ABB RobotStudio station: LAB1RS_20220902-140616.rsstn

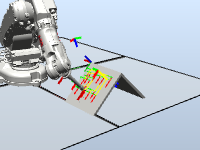
Station LAB1RS (saved by RobotStudio 6.5.7558.2005)
Controller IRB_140_6kg_0.81m
  mechanical unit ROB_1: IRB140_6_81_C_03, 6 joints, base frame (0, 0, 0) mm
Layout (positions relative to the parent item):
  - IRB140_6_81_C_03 [mechanism, from Robots\IRB140_6_81_C_G_03.rslib] at (0, 0, 0) mm; joint values [-0.1973, 1.0047, -0.2124, 0.8557, 1.1481, -2.2858] (rad or m)
  - TABLERO2 [part] at (800, 200, 0) mm, rotated rx 90 ry 0 rz 90 deg
  - TOOLSJ [mechanism, from Libraries\HCV2.rslib] at (628.25, -79.94, 228.26) mm, rotated rx 180 ry 44.6 rz -90 deg
Attachment: TOOLSJ is attached to IRB140_6_81_C_03 / Link6
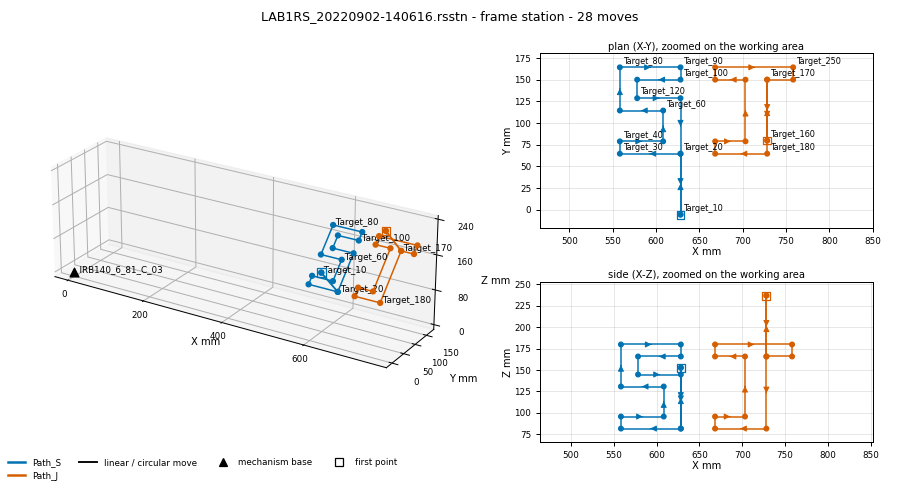
[picture p0: tool path of LAB1RS_20220902-140616.rsstn in frame station, 28 of 30 moves have a stored position in this frame; points joined in program order, loops and branches not executed]
Targets, tools, work objects and paths stored in the station, written as RAPID:
! task T_ROB1
MODULE CalibData
  TASK PERS wobjdata TabSJ:=[FALSE,TRUE,"",[[516.5,200,215],[0,0,-0.379480687,0.925199658]],[[0,0,0],[1,0,0,0]]];
  PERS tooldata HCVTCP:=[TRUE,[[0,0,191.01],[1,0,0,0]],[0.16,[0,0,75.29],[1,0,0,0],0,0,0]];
  PERS tooldata TOOLSJTCP:=[TRUE,[[0,0,191.01],[1,0,0,0]],[0.2,[0,0,1],[1,0,0,0],0,0,0]];
ENDMODULE

! task T_ROB1
MODULE Module1
  CONST jointtarget Home:=[[0,0,0,0,0,0],[9E+09,9E+09,9E+09,9E+09,9E+09,9E+09]];
  CONST jointtarget Mid:=[[0,30,0,0,30,0],[9E+09,9E+09,9E+09,9E+09,9E+09,9E+09]];
  CONST robtarget Target_10:=[[-111.75,190.000000035,99.999999935],[0,0.707106781,0.707106781,0],[0,0,0,0],[9E+09,9E+09,9E+09,9E+09,9E+09,9E+09]];
  CONST robtarget Target_20:=[[-111.75,190,-0.000000065],[0,0.707106781,0.707106781,0],[0,0,0,0],[9E+09,9E+09,9E+09,9E+09,9E+09,9E+09]];
  CONST robtarget Target_30:=[[-41.75,190,-0.000000065],[0,0.707106781,0.707106781,0],[0,0,0,0],[9E+09,9E+09,9E+09,9E+09,9E+09,9E+09]];
  CONST robtarget Target_40:=[[-41.75,170,-0.000000057],[0,0.707106781,0.707106781,0],[0,0,0,0],[9E+09,9E+09,9E+09,9E+09,9E+09,9E+09]];
  CONST robtarget Target_50:=[[-91.75,170,-0.000000057],[0,0.707106781,0.707106781,0],[0,0,0,0],[9E+09,9E+09,9E+09,9E+09,9E+09,9E+09]];
  CONST robtarget Target_60:=[[-91.75,120,-0.000000041],[0,0.707106781,0.707106781,0],[0,0,0,0],[9E+09,9E+09,9E+09,9E+09,9E+09,9E+09]];
  CONST robtarget Target_70:=[[-41.75,120,-0.000000041],[0,0.707106781,0.707106781,0],[0,0,0,0],[9E+09,9E+09,9E+09,9E+09,9E+09,9E+09]];
  CONST robtarget Target_80:=[[-41.75,50,-0.000000017],[0,0.707106781,0.707106781,0],[0,0,0,0],[9E+09,9E+09,9E+09,9E+09,9E+09,9E+09]];
  CONST robtarget Target_90:=[[-111.75,50,-0.000000017],[0,0.707106781,0.707106781,0],[0,0,0,0],[9E+09,9E+09,9E+09,9E+09,9E+09,9E+09]];
  CONST robtarget Target_100:=[[-111.75,70,-0.000000024],[0,0.707106781,0.707106781,0],[0,0,0,0],[9E+09,9E+09,9E+09,9E+09,9E+09,9E+09]];
  CONST robtarget Target_110:=[[-61.75,70,-0.000000024],[0,0.707106781,0.707106781,0],[0,0,0,0],[9E+09,9E+09,9E+09,9E+09,9E+09,9E+09]];
  CONST robtarget Target_120:=[[-61.75,100,-0.000000034],[0,0.707106781,0.707106781,0],[0,0,0,0],[9E+09,9E+09,9E+09,9E+09,9E+09,9E+09]];
  CONST robtarget Target_130:=[[-111.75,100,-0.000000034],[0,0.707106781,0.707106781,0],[0,0,0,0],[9E+09,9E+09,9E+09,9E+09,9E+09,9E+09]];
  CONST robtarget Target_140:=[[-111.75,190,-0.000000065],[0,0.707106781,0.707106781,0],[0,0,0,0],[9E+09,9E+09,9E+09,9E+09,9E+09,9E+09]];
  CONST robtarget Target_150:=[[-111.75,190.000000035,99.999999935],[0,0.707106781,0.707106781,0],[0,0,0,0],[9E+09,9E+09,9E+09,9E+09,9E+09,9E+09]];
  CONST robtarget Target_160:=[[-211.75,70.000000034,99.999999976],[0,0.707106781,0.707106781,0],[0,0,0,0],[9E+09,9E+09,9E+09,9E+09,9E+09,9E+09]];
  CONST robtarget Target_170:=[[-211.75,70,-0.000000024],[0,0.707106781,0.707106781,0],[0,0,0,0],[9E+09,9E+09,9E+09,9E+09,9E+09,9E+09]];
  CONST robtarget Target_180:=[[-211.75,190,-0.000000065],[0,0.707106781,0.707106781,0],[0,0,0,0],[9E+09,9E+09,9E+09,9E+09,9E+09,9E+09]];
  CONST robtarget Target_190:=[[-151.75,190,-0.000000065],[0,0.707106781,0.707106781,0],[0,0,0,0],[9E+09,9E+09,9E+09,9E+09,9E+09,9E+09]];
  CONST robtarget Target_200:=[[-151.75,170,-0.000000057],[0,0.707106781,0.707106781,0],[0,0,0,0],[9E+09,9E+09,9E+09,9E+09,9E+09,9E+09]];
  CONST robtarget Target_210:=[[-186.75,170,-0.000000057],[0,0.707106781,0.707106781,0],[0,0,0,0],[9E+09,9E+09,9E+09,9E+09,9E+09,9E+09]];
  CONST robtarget Target_220:=[[-186.75,70,-0.000000024],[0,0.707106781,0.707106781,0],[0,0,0,0],[9E+09,9E+09,9E+09,9E+09,9E+09,9E+09]];
  CONST robtarget Target_230:=[[-151.75,70,-0.000000024],[0,0.707106781,0.707106781,0],[0,0,0,0],[9E+09,9E+09,9E+09,9E+09,9E+09,9E+09]];
  CONST robtarget Target_240:=[[-151.75,50,-0.000000017],[0,0.707106781,0.707106781,0],[0,0,0,0],[9E+09,9E+09,9E+09,9E+09,9E+09,9E+09]];
  CONST robtarget Target_250:=[[-241.75,50,-0.000000017],[0,0.707106781,0.707106781,0],[0,0,0,0],[9E+09,9E+09,9E+09,9E+09,9E+09,9E+09]];
  CONST robtarget Target_260:=[[-241.75,70,-0.000000024],[0,0.707106781,0.707106781,0],[0,0,0,0],[9E+09,9E+09,9E+09,9E+09,9E+09,9E+09]];
  CONST robtarget Target_270:=[[-211.75,70,-0.000000024],[0,0.707106781,0.707106781,0],[0,0,0,0],[9E+09,9E+09,9E+09,9E+09,9E+09,9E+09]];
  CONST robtarget Target_280:=[[-211.75,70.000000034,99.999999976],[0,0.707106781,0.707106781,0],[0,0,0,0],[9E+09,9E+09,9E+09,9E+09,9E+09,9E+09]];
  PROC Path_S()
    MoveL Target_10,v200,z10,TOOLSJTCP\WObj:=TabSJ;
    MoveL Target_20,v200,z10,TOOLSJTCP\WObj:=TabSJ;
    MoveL Target_30,v200,z10,TOOLSJTCP\WObj:=TabSJ;
    MoveL Target_40,v200,z10,TOOLSJTCP\WObj:=TabSJ;
    MoveL Target_50,v200,z10,TOOLSJTCP\WObj:=TabSJ;
    MoveL Target_60,v200,z10,TOOLSJTCP\WObj:=TabSJ;
    MoveL Target_70,v200,z10,TOOLSJTCP\WObj:=TabSJ;
    MoveL Target_80,v200,z10,TOOLSJTCP\WObj:=TabSJ;
    MoveL Target_90,v200,z10,TOOLSJTCP\WObj:=TabSJ;
    MoveL Target_100,v200,z10,TOOLSJTCP\WObj:=TabSJ;
    MoveL Target_110,v200,z10,TOOLSJTCP\WObj:=TabSJ;
    MoveL Target_120,v200,z10,TOOLSJTCP\WObj:=TabSJ;
    MoveL Target_130,v200,z10,TOOLSJTCP\WObj:=TabSJ;
    MoveL Target_140,v200,z10,TOOLSJTCP\WObj:=TabSJ;
    MoveL Target_150,v200,z10,TOOLSJTCP\WObj:=TabSJ;
  ENDPROC
  PROC Path_J()
    MoveL Target_160,v200,z10,TOOLSJTCP\WObj:=TabSJ;
    MoveL Target_170,v200,z10,TOOLSJTCP\WObj:=TabSJ;
    MoveL Target_180,v200,z10,TOOLSJTCP\WObj:=TabSJ;
    MoveL Target_190,v200,z10,TOOLSJTCP\WObj:=TabSJ;
    MoveL Target_200,v200,z10,TOOLSJTCP\WObj:=TabSJ;
    MoveL Target_210,v200,z10,TOOLSJTCP\WObj:=TabSJ;
    MoveL Target_220,v200,z10,TOOLSJTCP\WObj:=TabSJ;
    MoveL Target_230,v200,z10,TOOLSJTCP\WObj:=TabSJ;
    MoveL Target_240,v200,z10,TOOLSJTCP\WObj:=TabSJ;
    MoveL Target_250,v200,z10,TOOLSJTCP\WObj:=TabSJ;
    MoveL Target_260,v200,z10,TOOLSJTCP\WObj:=TabSJ;
    MoveL Target_270,v200,z10,TOOLSJTCP\WObj:=TabSJ;
    MoveL Target_280,v200,z10,TOOLSJTCP\WObj:=TabSJ;
  ENDPROC
  PROC Path_H()
    MoveAbsJ Home,v400,z100,tool0\WObj:=TabSJ;
  ENDPROC
  PROC Path_M()
    MoveAbsJ Mid,v400,z100,tool0\WObj:=TabSJ;
  ENDPROC
ENDMODULE

